// TIA Portal V16 export
// export: Created 2023-08-28T09:37:54.3820337Z, ExportSetting WithDefaults, DisplayName Totally Integrated Automation Portal, DisplayVersion V16 Update 6, DisplayName TIA Portal Version Control Interface, DisplayVersion V16 Update 2, DisplayName TIA Portal Openness, DisplayVersion V16 Update 6, DisplayName STEP 7 Professional, DisplayVersion V16 Update 6, DisplayName STEP 7 Safety, DisplayVersion V16, DisplayName WinCC Advanced, DisplayVersion V16 Update 6
VAR_GLOBAL   // PLC tag table "P3"
   inputReadyP3 AT %M82.6 : Bool;   // sugnał gotowość / Gotowość napędu
   inputRunF_P3 AT %M82.7 : Bool;   // stycznik falownik / Potwierdzenie pracy z falownika
   inputRunS_P3 AT %M83.0 : Bool;   // stycznik softstart / Powierdzenie pracy z sieci
   CMD_inverter_P3 AT %M83.1 : Bool;   // Stycznik Falownik
   CMD_network_P3 AT %M83.2 : Bool;   // Stycznik Sieć
   setCMD_FP3 AT %M207.4 : Bool;   // Znacznik sterowania w trybie falownik dlaP1
   setCMD_SP3 AT %M207.5 : Bool;   // Znacznik sterowania w trybie sieć
   IsReady_P3 AT %M17.2 : Bool;   // Znacznik gotowości napędu
   CB_CMD_P3 AT %M12.6 : Bool;   // Znacznik polecenia on/off przekaźnik napędu
   Hour_Work_P3 AT %MD44 : DWord;   // Licznik pracy
   Set_HWork_P3 AT %M11.2 : Bool;   // Znacznik ustawienia aktywnej do pracy (po porównaniu liczników pracy)
   IsRunInverter_P3 AT %M211.5 : Bool;   // Potwierdzenie pracy z falownika
   IsRunNetwork_P3 AT %M217.2 : Bool;   // Potwierdzenie pracy z sieci
   Is_extras_K1_P3 AT %M218.6 : Bool;   // Znacznik motor dodatkowy nr 1
   Set_50Hz_P3 AT %M219.5 : Bool;   // Znacznik pamięci podtrzymujący przełączenie na sieć
   setSUPV_FP3 AT %M12.2 : Bool;   // Znacznik polecenia startu z falownika
   IsRun_P3 AT %M11.6 : Bool;   // Potwierdzenie pracy
   setSUPV_SP3 AT %M13.1 : Bool;   // Znacznik polecenia startu z sieci
   CMD_soft_P3 AT %M85.1 : Bool;   // sygnał z softstart potwierdzenie pracy / sygnał on/off soft-start
   resetFault_SoftStart_P3 AT %M50.2 : Bool;   // sygnał resetu softstart
   bitH_REM_P3 AT %M64.2 : Bool;   // Zdalna - kopia bitu z instancji statusu napędu
   bitH_RUN_P3 AT %M64.3 : Bool;   // Praca - kopia bitu z instancji statusu napędu
   bitH_OFF_P3 AT %M64.4 : Bool;   // Polecenie OFF - kopia bitu z instancji statusu napędu
   bitH_ON_P3 AT %M64.5 : Bool;   // Polecenie ON - kopia bitu z instancji statusu napędu
   bitH_Res_P3 AT %M64.6 : Bool;   // Reset - kopia bitu z instancji statusu napędu
   bitH_Aut_Man_P3 AT %M64.7 : Bool;   // Aut=1 Man=0 - kopia bitu z instancji statusu napędu
   bitH_Alarm_P3 AT %M64.0 : Bool;   // Alarm - kopia bitu z instancji statusu napędu
   bitH_rezerwa_P3 AT %M64.1 : Bool;   // rez
   Is_extras_K3_P3 AT %M89.7 : Bool;   // Znacznik motor dodatkowy nr 3
   Is_extras_K2_P3 AT %M219.1 : Bool;   // Znacznik motor dodatkowy nr 2
   off_add_K1_P3 AT %M52.6 : Bool;   // sterowanie wyłączeniem selektywnym dodatkowej
   off_add_K2_P3 AT %M52.7 : Bool;   // sterowanie wyłączeniem selektywnym dodatkowej
   off_add_K3_P3 AT %M53.0 : Bool;   // sterowanie wyłączeniem selektywnym dodatkowej
   off_add_K4_P3 AT %M53.6 : Bool;   // sterowanie wyłączeniem selektywnym dodatkowej
   CMD_ErrorSet_NetworkM3 AT %M221.5 : Bool;   // Znacznik sterowania awaryjnego pracą pompy bez falownika
   Mem_Res_setCMD_MC_P3 AT %M223.2 : Bool;   // pamięć zbocza załączenia timera blokowania stycznika falowni
END_VAR
